// TIA Portal V19 export
DATA_BLOCK "OP25 TANK"   // DB42
{ S7_Optimized_Access := 'TRUE' }
AUTHOR : OPA_8160
FAMILY : APP
NAME : OP25
// stored: AutoNumber false, MemoryReserve 0
   VAR RETAIN
      TaTimerStep : S5Time;
      TaTimerActual : S5Time;
      TaMainUpdating : Int := 6;
      TaStepUpdating : Int := 161;
      TaRcNoUpdating : Int := 4;   // RECIPE NO. UPDATING,NOT USED IN TANK-PLC
      TaRcNoEntering : Int := 4;   // RECIPE NO. ENTERING,NOT USED IN TANK-PLC
      TaPointerRcDB : Int := 51;   // CONTAINS DB NO FOR RECIPE,NOT USED IN TANK-PLC
      FilTimerStep : S5Time;
      FilTimerActual : S5Time;
      FilMainUpdating : Int;
      FilStepUpdating : Int;
      Reset_lamp_Scada : Bool;   // Reset bit from Scada
      TIM_STP_INTOUCH : Int;   // Actual timer setpoint to intouch
      TIM_ACT_INTOUCH : Int;   // Actual timer value to intouch
      RuninghoursAHV : Real := 18205.97;
   END_VAR
BEGIN
END_DATA_BLOCK
